TYPE "UDT_ZC_COM_REAL"
VERSION : 0.1
   STRUCT
      In : Real;
      Out : Real;
      Forzar : Bool;   // 0= Automatico / 1= Forzado
      ValorForzado : Real;   // Valor forzado
   END_STRUCT;

END_TYPE

